{attribute 'pack_mode' := '1'}
TYPE ST_SystemSettingsReport :
STRUCT
	sGenSealAndPump               : STRING(100);
    sCalAcceptanceCriteria        : STRING(100);
    sCalAllowableFail             : STRING(100);
    sCalReplicates                : STRING(100);
    sCalPumpCallIntervalDays      : STRING(100);
    sCalCloseAppOnCompletion      : STRING(100);
    sAirDryTimeOnCompletion       : STRING(100);
    sLktAllowableLeakTestFail     : STRING(100);
    sLktLeakTestBuildUpTime       : STRING(100);
    sLktLeakTestHoldTime          : STRING(100);
    sLktLeakTestPressure          : STRING(100);
    sMecPlatesClosedPosition      : STRING(100);
    sMecPlatesDryPosition         : STRING(100);
    sMecPlatesVelocity            : STRING(100);
    sMecMaxCurrentFastDown        : STRING(100);
    sMecMaxCurrentSlowDown        : STRING(100);
    sMecMaxCurrentSlowUp          : STRING(100);
    sPmpMeterVelocity             : STRING(100);
    sPmpRunVelocity               : STRING(100);
    sPmpEmptyFactor               : STRING(100);
    sPmpFillSolventTubesFactor    : STRING(100);
    sSmpAboveCalibration          : STRING(100);
    sSmpVialSetSpacing            : STRING(100);
    sSmpIntoResBottom             : STRING(100);
    sSmpIntoResDispense           : STRING(100);
    sSmpIntoResWeigh              : STRING(100);
    sSmpIntoVials                 : STRING(100);
    sSmpIntoWaste                 : STRING(100);
    sSecDisplayManualControl      : STRING(100);
    sSecCheckLogonEachRun         : STRING(100);
    sCreatedBy                    : STRING(100);
    sCreatedDate                  : STRING(100);
    sSysRevisionNo                : STRING(30);
END_STRUCT
END_TYPE

(* stored: Version 1.1.0.1, ProductVersion 3.1.4024.15
   DUT ST_SystemSettingsReport: Id {619a8ab0-d2f0-480d-9f07-bfccdda7aa59} *)
